(* PLC project Unnamed, Unknown Unnamed 1 *)
(* stored: creationDateTime 2026-05-13T00:02:20, modificationDateTime 2026-05-13T00:02:20 *)

FUNCTION_BLOCK Test
  VAR_INPUT
    Input : BOOL;
  END_VAR
  VAR_OUTPUT
    Output : BOOL;
  END_VAR

            Output := Input;
          
END_FUNCTION_BLOCK

PROGRAM main
  VAR
    Input0 AT %IX0.0 : BOOL;
    Output0 AT %QX0.0 : BOOL;
  END_VAR
  VAR
    TestFunktion : TEST;
  END_VAR

            TestFunktion(
    Input := Input0
);

Output0 := TestFunktion.Output or true;
          
END_PROGRAM

CONFIGURATION Config0
  RESOURCE Res0 ON PLC
    TASK task0(INTERVAL := T#10ms, PRIORITY := 1);
    PROGRAM instance0 WITH task0 : main;
  END_RESOURCE
END_CONFIGURATION
